{attribute 'qualified_only'}
{attribute 'strict'}
{attribute 'to_string'}
TYPE E_MachineState :
(
	INITIALIZATION	:= 0,
	RUN 			:= 1,
	HOLD 			:= 2,
	ERROR	 		:= 3,
	RESET			:= 4,
	TOOLCALIBRATION := 5,
	TOOLCHANGERUN	:= 6,
	TOOLCHANGEINIT 	:= 7,
	RUNMANUAL		:= 8
);
END_TYPE

(* stored: Version 1.1.0.1, ProductVersion 3.1.4024.12
   EnumerationTextList E_MachineState: Id {580642a0-2ba0-4ed4-877e-7b89e74756f9} *)
